# EPICS autosave request: dxpApp/Db/dxpMED_settings.req
$(P)PresetMode
$(P)PresetReal
$(P)PresetEvents
$(P)PresetTriggers
$(P)StatusAll.SCAN
$(P)ReadAll.SCAN
$(P)TraceTimes
$(P)EnableClientWait
